(* Schneider Machine Expert - Basic project SORTING_3_WAY_TM221CE24R_REV3, file version 3.0.0.0 *)
(* ProjectInformations: Name=New project *)

HARDWARE
  Cpu 0: TM221CE24R
  ModuleExtensionObject 0: TM3DI32K
  ModuleExtensionObject 1: TM3AI2H/G
  EthernetConfiguration: NetworkName=M221, IpAllocationMode=FixedAddress, IpAddress=0.0.0.0, SubnetMask=0.0.0.0
  SerialLineConfiguration: Baud=Baud19200, Parity=ParityEven, DataBits=DataBits8, StopBits=StopBits1, PhysicalMedium=PhysicalMediumRs485, TransmissionMode=TransmissionModeModbusRtu, SlaveId=1, Addressing=SlaveAddressing
  MastTask: UsePeriodScanMode=false, PeriodScan=100
  FastTask: Period=255
  CpuBehavior: StartingMode=StartAsPreviousState, AutoSaveRamOnEeprom=true, WatchdogPeriod=250

SYMBOLS  (address, symbol, comment, settings)
  %M0       AUTO_MODE  "1 Auto"
  %M1       START_HMI  "Start HMI momentary"
  %M2       STOP_HMI  "Stop HMI"
  %M3       AUTO_ENABLE  "Izin auto"
  %M10      RUN_MEMORY  "Latch produksi"
  %M11      SAFETY_OK  "Ringkasan interlock"
  %M20      PRODUCT_A_LATCH  "Produk A"
  %M21      PRODUCT_B_LATCH  "Produk B"
  %M22      PRODUCT_REJECT_LATCH  "Produk reject"
  %M23      SORT_BUSY  "Sequence sortir aktif"
  %M24      TRANSPORT_DONE  "Produk sampai aktuator"
  %M25      PUSH_ACTIVE  "Aktuator sortir aktif"
  %M26      PUSH_DONE  "Pulsa selesai pusher"
  %M27      EXIT_PULSE  "Pulsa satu scan sensor keluar"
  %M30      JAM_ALARM_LATCH  "Timeout sortir"
  %M31      BIN_ALARM_LATCH  "Reject bin penuh"
  %M32      ALARM_ACTIVE  "Alarm umum"
  %M40      RESET_HMI  "Reset HMI"
  %M41      RESET_COUNTERS_HMI  "Reset production counter"
  %M42      RESET_REQUEST  "Gabungan reset"
  %S5       SB_TB100MS  "Time base of 100 ms generated by an internal clock"
  %S6       SB_TB1S  "Time base of 1 s generated by an internal clock"
  %S13      SB_FIRSTRUN  "Indicates the first controller cycle in RUN mode"
  %MW1      WATER_RANGE_MM  "Range sensor level mm"
  %MW2      LEVEL_RAW_COPY  "Salinan raw input level"
  %MW10     MAX_HEIGHT_G1_MM  "Tinggi maksimum pintu 1 mm"
  %MW11     MAX_HEIGHT_G2_MM  "Tinggi maksimum pintu 2 mm"
  %MW12     MAX_HEIGHT_G3_MM  "Tinggi maksimum pintu 3 mm"
  %MW13     DEADBAND_PCT  "Deadband posisi persen"
  %MW20     ENC_ZERO_G1  "Nilai encoder pintu 1 saat tertutup"
  %MW21     ENC_ZERO_G2  "Nilai encoder pintu 2 saat tertutup"
  %MW22     ENC_ZERO_G3  "Nilai encoder pintu 3 saat tertutup"
  %MW23     ENC_SPAN_G1  "Span count tertutup-terbuka G1"
  %MW24     ENC_SPAN_G2  "Span count tertutup-terbuka G2"
  %MW25     ENC_SPAN_G3  "Span count tertutup-terbuka G3"
  %MW30     ENC_BINARY_G1  "Nilai biner encoder G1"
  %MW31     ENC_BINARY_G2  "Nilai biner encoder G2"
  %MW32     ENC_BINARY_G3  "Nilai biner encoder G3"
  %MW33     POS_COUNT_G1  "Count posisi terkoreksi G1"
  %MW34     POS_COUNT_G2  "Count posisi terkoreksi G2"
  %MW35     POS_COUNT_G3  "Count posisi terkoreksi G3"
  %MW50     TARGET_PCT_G1  "Target bukaan G1 0-100 persen"
  %MW51     TARGET_PCT_G2  "Target bukaan G2 0-100 persen"
  %MW52     TARGET_PCT_G3  "Target bukaan G3 0-100 persen"
  %MF60     POSITION_G1_PCT  "Posisi G1 persen"
  %MF62     POSITION_G2_PCT  "Posisi G2 persen"
  %MF64     POSITION_G3_PCT  "Posisi G3 persen"
  %MF66     POSITION_G1_MM  "Posisi G1 mm"
  %MF68     POSITION_G2_MM  "Posisi G2 mm"
  %MF70     POSITION_G3_MM  "Posisi G3 mm"
  %MF72     WATER_LEVEL_MM  "Level air mm"
  %MF74     WATER_LEVEL_PCT  "Level air persen"
  %MF76     WATER_RANGE_REAL  "Range level dalam REAL"
  %MF80     TARGET_G1_REAL  "Target G1 dalam REAL"
  %MF82     TARGET_G2_REAL  "Target G2 dalam REAL"
  %MF84     TARGET_G3_REAL  "Target G3 dalam REAL"
  %MF86     DEADBAND_REAL  "Deadband dalam REAL"
  %MF88     OPEN_THRESHOLD_G1  "Ambang buka G1"
  %MF90     CLOSE_THRESHOLD_G1  "Ambang tutup G1"
  %MF92     OPEN_THRESHOLD_G2  "Ambang buka G2"
  %MF94     CLOSE_THRESHOLD_G2  "Ambang tutup G2"
  %MF96     OPEN_THRESHOLD_G3  "Ambang buka G3"
  %MF98     CLOSE_THRESHOLD_G3  "Ambang tutup G3"
  %C0       TRANSPORT_TICKS  "20 x pulsa 100 ms = 2 s"
  %C1       PUSH_TICKS  "7 x pulsa 100 ms = 0.7 s"
  %C2       SEQUENCE_SECONDS  "8 x pulsa 1 s = timeout 8 s"
  %C3       COUNT_A  "Jumlah produk A"
  %C4       COUNT_B  "Jumlah produk B"
  %C5       COUNT_REJECT  "Jumlah produk reject"
  %I0.0     START_PB  "Tombol Start NO"
  %I0.1     STOP_OK  "Kontak Stop NC; 1 sehat"
  %I0.2     ESTOP_OK  "Feedback safety relay; 1 sehat"
  %I0.3     OVERLOAD_OK  "Overload conveyor; 1 sehat"
  %I0.4     ENTRY_SENSOR  "Sensor produk masuk"
  %I0.5     TYPE_A_SENSOR  "Sensor klasifikasi A"
  %I0.6     TYPE_B_SENSOR  "Sensor klasifikasi B"
  %I0.7     PUSHER_HOME  "Pusher pada posisi home"
  %I0.8     EXIT_SENSOR  "Sensor keluar"
  %I0.9     BIN_A_AVAILABLE  "Bin A belum penuh"
  %I0.10    BIN_B_AVAILABLE  "Bin B belum penuh"
  %I0.11    REJECT_BIN_AVAILABLE  "Bin reject belum penuh"
  %I0.12    RESET_PB  "Reset alarm"
  %I0.13      "Tidak digunakan"
  %Q0.0     MOTOR_CONVEYOR  "Kontaktor/VFD conveyor"
  %Q0.1     PUSHER_A  "Solenoid pusher A"
  %Q0.2     PUSHER_B  "Solenoid pusher B"
  %Q0.3     REJECT_GATE  "Solenoid gate reject"
  %Q0.4     LAMP_RUN  "Lampu run"
  %Q0.5     LAMP_BUSY  "Lampu sequence busy"
  %Q0.6     LAMP_FAULT  "Lampu fault"
  %Q0.7     BUZZER  "Buzzer fault"
  %Q0.8       "Tidak digunakan"
  %Q0.9       "Tidak digunakan"
  %I1.0     ENC_G1_GRAY_B0  "E6CP pintu 1 Gray bit 0"
  %I1.1     ENC_G1_GRAY_B1  "E6CP pintu 1 Gray bit 1"
  %I1.2     ENC_G1_GRAY_B2  "E6CP pintu 1 Gray bit 2"
  %I1.3     ENC_G1_GRAY_B3  "E6CP pintu 1 Gray bit 3"
  %I1.4     ENC_G1_GRAY_B4  "E6CP pintu 1 Gray bit 4"
  %I1.5     ENC_G1_GRAY_B5  "E6CP pintu 1 Gray bit 5"
  %I1.6     ENC_G1_GRAY_B6  "E6CP pintu 1 Gray bit 6"
  %I1.7     ENC_G1_GRAY_B7  "E6CP pintu 1 Gray bit 7"
  %I1.8     ENC_G2_GRAY_B0  "E6CP pintu 2 Gray bit 0"
  %I1.9     ENC_G2_GRAY_B1  "E6CP pintu 2 Gray bit 1"
  %I1.10    ENC_G2_GRAY_B2  "E6CP pintu 2 Gray bit 2"
  %I1.11    ENC_G2_GRAY_B3  "E6CP pintu 2 Gray bit 3"
  %I1.12    ENC_G2_GRAY_B4  "E6CP pintu 2 Gray bit 4"
  %I1.13    ENC_G2_GRAY_B5  "E6CP pintu 2 Gray bit 5"
  %I1.14    ENC_G2_GRAY_B6  "E6CP pintu 2 Gray bit 6"
  %I1.15    ENC_G2_GRAY_B7  "E6CP pintu 2 Gray bit 7"
  %I1.16    ENC_G3_GRAY_B0  "E6CP pintu 3 Gray bit 0"
  %I1.17    ENC_G3_GRAY_B1  "E6CP pintu 3 Gray bit 1"
  %I1.18    ENC_G3_GRAY_B2  "E6CP pintu 3 Gray bit 2"
  %I1.19    ENC_G3_GRAY_B3  "E6CP pintu 3 Gray bit 3"
  %I1.20    ENC_G3_GRAY_B4  "E6CP pintu 3 Gray bit 4"
  %I1.21    ENC_G3_GRAY_B5  "E6CP pintu 3 Gray bit 5"
  %I1.22    ENC_G3_GRAY_B6  "E6CP pintu 3 Gray bit 6"
  %I1.23    ENC_G3_GRAY_B7  "E6CP pintu 3 Gray bit 7"
  %I1.24    MODE_AUTO  "Selector 1=AUTO 0=MANUAL"
  %I1.25    MAN_OPEN_G1  "PB manual buka pintu 1"
  %I1.26    MAN_CLOSE_G1  "PB manual tutup pintu 1"
  %I1.27    MAN_OPEN_G2  "PB manual buka pintu 2"
  %I1.28    MAN_CLOSE_G2  "PB manual tutup pintu 2"
  %I1.29    MAN_OPEN_G3  "PB manual buka pintu 3"
  %I1.30    MAN_CLOSE_G3  "PB manual tutup pintu 3"
  %I1.31    RESET_FAULT  "PB reset fault"
  %IW2.0    LEVEL_RAW  "Sensor level 4-20 mA raw 4000-20000"  [Type=Type_4_20mA, Scope=Scope_Customized, Minimum=4000, Maximum=20000]

POU SORTING_3_WAY_IL
  (* SectionNumber=1 *)

// Rung 0: N01_SAFETY
// Safety feedback.
  LD %I0.1                (* STOP_OK *)
  AND %I0.2               (* ESTOP_OK *)
  AND %I0.3               (* OVERLOAD_OK *)
  ANDN %M2                (* STOP_HMI *)
  ST %M11                 (* SAFETY_OK *)
  // as ST:
  //   SAFETY_OK := STOP_OK AND ESTOP_OK AND OVERLOAD_OK AND NOT STOP_HMI;

// Rung 1: N02_RUN
// Latch auto run.
  LD %I0.0                (* START_PB *)
  OR %M1                  (* START_HMI *)
  OR %M10                 (* RUN_MEMORY *)
  AND %M0                 (* AUTO_MODE *)
  AND %M3                 (* AUTO_ENABLE *)
  AND %M11                (* SAFETY_OK *)
  ST %M10                 (* RUN_MEMORY *)
  // as ST:
  //   RUN_MEMORY := (START_PB OR START_HMI OR RUN_MEMORY) AND AUTO_MODE AND AUTO_ENABLE AND SAFETY_OK;

// Rung 2: N03_RESET
// Gabungan reset.
  LD %I0.12               (* RESET_PB *)
  OR %M40                 (* RESET_HMI *)
  ST %M42                 (* RESET_REQUEST *)
  // as ST:
  //   RESET_REQUEST := RESET_PB OR RESET_HMI;

// Rung 3: N04_CLASS_A
// Tangkap produk A.
  LDR %I0.4               (* ENTRY_SENSOR *)
  AND %M10                (* RUN_MEMORY *)
  ANDN %M23               (* SORT_BUSY *)
  AND %I0.5               (* TYPE_A_SENSOR *)
  AND %I0.9               (* BIN_A_AVAILABLE *)
  S %M20                  (* PRODUCT_A_LATCH *)
  // as ST:
  //   IF RISING(ENTRY_SENSOR) AND RUN_MEMORY AND NOT SORT_BUSY AND TYPE_A_SENSOR AND BIN_A_AVAILABLE THEN PRODUCT_A_LATCH := TRUE; END_IF;

// Rung 4: N05_CLASS_B
// Tangkap produk B.
  LDR %I0.4               (* ENTRY_SENSOR *)
  AND %M10                (* RUN_MEMORY *)
  ANDN %M23               (* SORT_BUSY *)
  ANDN %I0.5              (* TYPE_A_SENSOR *)
  AND %I0.6               (* TYPE_B_SENSOR *)
  AND %I0.10              (* BIN_B_AVAILABLE *)
  S %M21                  (* PRODUCT_B_LATCH *)
  // as ST:
  //   IF RISING(ENTRY_SENSOR) AND RUN_MEMORY AND NOT SORT_BUSY AND NOT TYPE_A_SENSOR AND TYPE_B_SENSOR AND BIN_B_AVAILABLE THEN PRODUCT_B_LATCH := TRUE; END_IF;

// Rung 5: N06_CLASS_REJECT
// Selain A/B masuk reject.
  LDR %I0.4               (* ENTRY_SENSOR *)
  AND %M10                (* RUN_MEMORY *)
  ANDN %M23               (* SORT_BUSY *)
  ANDN %M20               (* PRODUCT_A_LATCH *)
  ANDN %M21               (* PRODUCT_B_LATCH *)
  AND %I0.11              (* REJECT_BIN_AVAILABLE *)
  S %M22                  (* PRODUCT_REJECT_LATCH *)
  // as ST:
  //   IF RISING(ENTRY_SENSOR) AND RUN_MEMORY AND NOT SORT_BUSY AND NOT PRODUCT_A_LATCH AND NOT PRODUCT_B_LATCH AND REJECT_BIN_AVAILABLE THEN PRODUCT_REJECT_LATCH := TRUE; END_IF;

// Rung 6: N07_BIN_FULL
// Alarm jika reject dibutuhkan tetapi bin penuh.
  LDR %I0.4               (* ENTRY_SENSOR *)
  AND %M10                (* RUN_MEMORY *)
  ANDN %M23               (* SORT_BUSY *)
  ANDN %M20               (* PRODUCT_A_LATCH *)
  ANDN %M21               (* PRODUCT_B_LATCH *)
  ANDN %I0.11             (* REJECT_BIN_AVAILABLE *)
  S %M31                  (* BIN_ALARM_LATCH *)
  // as ST:
  //   IF RISING(ENTRY_SENSOR) AND RUN_MEMORY AND NOT SORT_BUSY AND NOT PRODUCT_A_LATCH AND NOT PRODUCT_B_LATCH AND NOT REJECT_BIN_AVAILABLE THEN BIN_ALARM_LATCH := TRUE; END_IF;

// Rung 7: N08_SORT_BUSY
// Mulai sequence.
  LD %M20                 (* PRODUCT_A_LATCH *)
  OR %M21                 (* PRODUCT_B_LATCH *)
  OR %M22                 (* PRODUCT_REJECT_LATCH *)
  S %M23                  (* SORT_BUSY *)
  // as ST:
  //   IF PRODUCT_A_LATCH OR PRODUCT_B_LATCH OR PRODUCT_REJECT_LATCH THEN SORT_BUSY := TRUE; END_IF;

// Rung 8: N09_PRESET_C0
// Preset transport saat first scan.
  LD %S13                 (* SB_FIRSTRUN *)
  [ %C0.P := 20 ]         (* TRANSPORT_TICKS *)
  // as ST:
  //   IF SB_FIRSTRUN THEN TRANSPORT_TICKS.P := 20; END_IF;

// Rung 9: N09_PRESET_C1
// Preset pusher saat first scan.
  LD %S13                 (* SB_FIRSTRUN *)
  [ %C1.P := 7 ]          (* PUSH_TICKS *)
  // as ST:
  //   IF SB_FIRSTRUN THEN PUSH_TICKS.P := 7; END_IF;

// Rung 10: N09_PRESET_C2
// Preset timeout saat first scan.
  LD %S13                 (* SB_FIRSTRUN *)
  [ %C2.P := 8 ]          (* SEQUENCE_SECONDS *)
  // as ST:
  //   IF SB_FIRSTRUN THEN SEQUENCE_SECONDS.P := 8; END_IF;

// Rung 11: N10_TRANSPORT_COUNTER
// Hitung 2 detik menuju aktuator.
  BLK %C0                 (* TRANSPORT_TICKS *)
  LD %S5                  (* SB_TB100MS *)
  AND %M23                (* SORT_BUSY *)
  ANDN %M24               (* TRANSPORT_DONE *)
  CU
  LDN %M23                (* SORT_BUSY *)
  OR %M24                 (* TRANSPORT_DONE *)
  R
  END_BLK
  // as ST:
  //   TRANSPORT_TICKS(CU := SB_TB100MS AND SORT_BUSY AND NOT TRANSPORT_DONE, R := NOT SORT_BUSY OR TRANSPORT_DONE);

// Rung 12: N11_AT_POSITION
// Aktifkan pusher bila home.
  LD %C0.D                (* TRANSPORT_TICKS *)
  AND %I0.7               (* PUSHER_HOME *)
  S %M24                  (* TRANSPORT_DONE *)
  S %M25                  (* PUSH_ACTIVE *)
  // as ST:
  //   IF TRANSPORT_TICKS.D AND PUSHER_HOME THEN TRANSPORT_DONE := TRUE; END_IF;
  //   IF TRANSPORT_TICKS.D AND PUSHER_HOME THEN PUSH_ACTIVE := TRUE; END_IF;

// Rung 13: N13_PUSH_COUNTER
// Durasi aktuator 0.7 detik.
  BLK %C1                 (* PUSH_TICKS *)
  LD %S5                  (* SB_TB100MS *)
  AND %M25                (* PUSH_ACTIVE *)
  CU
  LDN %M25                (* PUSH_ACTIVE *)
  R
  END_BLK
  // as ST:
  //   PUSH_TICKS(CU := SB_TB100MS AND PUSH_ACTIVE, R := NOT PUSH_ACTIVE);

// Rung 14: N14_PUSH_DONE
// Akhiri aktuator.
  LD %C1.D                (* PUSH_TICKS *)
  ST %M26                 (* PUSH_DONE *)
  R %M25                  (* PUSH_ACTIVE *)
  // as ST:
  //   PUSH_DONE := PUSH_TICKS.D;
  //   IF PUSH_TICKS.D THEN PUSH_ACTIVE := FALSE; END_IF;

// Rung 15: N16_TIMEOUT_COUNTER
// Hitung maksimum waktu sequence.
  BLK %C2                 (* SEQUENCE_SECONDS *)
  LD %S6                  (* SB_TB1S *)
  AND %M23                (* SORT_BUSY *)
  CU
  LDN %M23                (* SORT_BUSY *)
  R
  END_BLK
  // as ST:
  //   SEQUENCE_SECONDS(CU := SB_TB1S AND SORT_BUSY, R := NOT SORT_BUSY);

// Rung 16: N17_TIMEOUT_ALARM
// Latch timeout.
  LD %C2.D                (* SEQUENCE_SECONDS *)
  S %M30                  (* JAM_ALARM_LATCH *)
  // as ST:
  //   IF SEQUENCE_SECONDS.D THEN JAM_ALARM_LATCH := TRUE; END_IF;

// Rung 17: N18_EXIT_PULSE
// Pulsa produk selesai.
  LDR %I0.8               (* EXIT_SENSOR *)
  AND %M23                (* SORT_BUSY *)
  ST %M27                 (* EXIT_PULSE *)
  // as ST:
  //   EXIT_PULSE := RISING(EXIT_SENSOR) AND SORT_BUSY;

// Rung 18: N19_COUNT_A
// Counter produksi A.
  BLK %C3                 (* COUNT_A *)
  LD %M27                 (* EXIT_PULSE *)
  AND %M20                (* PRODUCT_A_LATCH *)
  CU
  LD %M41                 (* RESET_COUNTERS_HMI *)
  R
  END_BLK
  // as ST:
  //   COUNT_A(CU := EXIT_PULSE AND PRODUCT_A_LATCH, R := RESET_COUNTERS_HMI);

// Rung 19: N20_COUNT_B
// Counter produksi B.
  BLK %C4                 (* COUNT_B *)
  LD %M27                 (* EXIT_PULSE *)
  AND %M21                (* PRODUCT_B_LATCH *)
  CU
  LD %M41                 (* RESET_COUNTERS_HMI *)
  R
  END_BLK
  // as ST:
  //   COUNT_B(CU := EXIT_PULSE AND PRODUCT_B_LATCH, R := RESET_COUNTERS_HMI);

// Rung 20: N21_COUNT_REJECT
// Counter produk reject.
  BLK %C5                 (* COUNT_REJECT *)
  LD %M27                 (* EXIT_PULSE *)
  AND %M22                (* PRODUCT_REJECT_LATCH *)
  CU
  LD %M41                 (* RESET_COUNTERS_HMI *)
  R
  END_BLK
  // as ST:
  //   COUNT_REJECT(CU := EXIT_PULSE AND PRODUCT_REJECT_LATCH, R := RESET_COUNTERS_HMI);

// Rung 21: N22_CLEAR_SEQUENCE
// Bersihkan latch setelah exit.
  LD %M27                 (* EXIT_PULSE *)
  R %M25                  (* PUSH_ACTIVE *)
  R %M24                  (* TRANSPORT_DONE *)
  R %M23                  (* SORT_BUSY *)
  R %M20                  (* PRODUCT_A_LATCH *)
  R %M21                  (* PRODUCT_B_LATCH *)
  R %M22                  (* PRODUCT_REJECT_LATCH *)
  // as ST:
  //   IF EXIT_PULSE THEN PUSH_ACTIVE := FALSE; END_IF;
  //   IF EXIT_PULSE THEN TRANSPORT_DONE := FALSE; END_IF;
  //   IF EXIT_PULSE THEN SORT_BUSY := FALSE; END_IF;
  //   IF EXIT_PULSE THEN PRODUCT_A_LATCH := FALSE; END_IF;
  //   IF EXIT_PULSE THEN PRODUCT_B_LATCH := FALSE; END_IF;
  //   IF EXIT_PULSE THEN PRODUCT_REJECT_LATCH := FALSE; END_IF;

// Rung 22: N23_RESET_JAM
// Reset timeout setelah kondisi pulih.
  LD %M42                 (* RESET_REQUEST *)
  ANDN %I0.4              (* ENTRY_SENSOR *)
  AND %I0.7               (* PUSHER_HOME *)
  R %M30                  (* JAM_ALARM_LATCH *)
  // as ST:
  //   IF RESET_REQUEST AND NOT ENTRY_SENSOR AND PUSHER_HOME THEN JAM_ALARM_LATCH := FALSE; END_IF;

// Rung 23: N24_RESET_BIN
// Reset bin alarm setelah tersedia.
  LD %M42                 (* RESET_REQUEST *)
  AND %I0.11              (* REJECT_BIN_AVAILABLE *)
  R %M31                  (* BIN_ALARM_LATCH *)
  // as ST:
  //   IF RESET_REQUEST AND REJECT_BIN_AVAILABLE THEN BIN_ALARM_LATCH := FALSE; END_IF;

// Rung 24: N25_ALARM
// Ringkasan alarm.
  LD %M30                 (* JAM_ALARM_LATCH *)
  OR %M31                 (* BIN_ALARM_LATCH *)
  ORN %I0.2               (* ESTOP_OK *)
  ORN %I0.3               (* OVERLOAD_OK *)
  ST %M32                 (* ALARM_ACTIVE *)
  // as ST:
  //   ALARM_ACTIVE := JAM_ALARM_LATCH OR BIN_ALARM_LATCH OR NOT ESTOP_OK OR NOT OVERLOAD_OK;

// Rung 25: N26_MOTOR
// Motor berhenti saat pusher/alarm.
  LD %M10                 (* RUN_MEMORY *)
  AND %M11                (* SAFETY_OK *)
  ANDN %M25               (* PUSH_ACTIVE *)
  ANDN %M32               (* ALARM_ACTIVE *)
  ST %Q0.0                (* MOTOR_CONVEYOR *)
  // as ST:
  //   MOTOR_CONVEYOR := RUN_MEMORY AND SAFETY_OK AND NOT PUSH_ACTIVE AND NOT ALARM_ACTIVE;

// Rung 26: N27_PUSHER_A
// Output A.
  LD %M25                 (* PUSH_ACTIVE *)
  AND %M20                (* PRODUCT_A_LATCH *)
  AND %M11                (* SAFETY_OK *)
  ST %Q0.1                (* PUSHER_A *)
  // as ST:
  //   PUSHER_A := PUSH_ACTIVE AND PRODUCT_A_LATCH AND SAFETY_OK;

// Rung 27: N28_PUSHER_B
// Output B.
  LD %M25                 (* PUSH_ACTIVE *)
  AND %M21                (* PRODUCT_B_LATCH *)
  AND %M11                (* SAFETY_OK *)
  ST %Q0.2                (* PUSHER_B *)
  // as ST:
  //   PUSHER_B := PUSH_ACTIVE AND PRODUCT_B_LATCH AND SAFETY_OK;

// Rung 28: N29_REJECT
// Output reject.
  LD %M25                 (* PUSH_ACTIVE *)
  AND %M22                (* PRODUCT_REJECT_LATCH *)
  AND %M11                (* SAFETY_OK *)
  ST %Q0.3                (* REJECT_GATE *)
  // as ST:
  //   REJECT_GATE := PUSH_ACTIVE AND PRODUCT_REJECT_LATCH AND SAFETY_OK;

// Rung 29: N30_LAMP_RUN
// Lampu run.
  LD %M10                 (* RUN_MEMORY *)
  ANDN %M32               (* ALARM_ACTIVE *)
  ST %Q0.4                (* LAMP_RUN *)
  // as ST:
  //   LAMP_RUN := RUN_MEMORY AND NOT ALARM_ACTIVE;

// Rung 30: N31_LAMP_BUSY
// Lampu sequence busy.
  LD %M23                 (* SORT_BUSY *)
  ST %Q0.5                (* LAMP_BUSY *)
  // as ST:
  //   LAMP_BUSY := SORT_BUSY;

// Rung 31: N32_FAULT_OUTPUTS
// Lampu fault dan buzzer.
  LD %M32                 (* ALARM_ACTIVE *)
  ST %Q0.6                (* LAMP_FAULT *)
  ST %Q0.7                (* BUZZER *)
  // as ST:
  //   LAMP_FAULT := ALARM_ACTIVE;
  //   BUZZER := ALARM_ACTIVE;
